FUNCTION TryConvert_USINT_TO_DWORD : BOOL
VAR_INPUT
	in : USINT;
	out : REFERENCE TO DWORD;
END_VAR

out := USINT_TO_DWORD(in);
TryConvert_USINT_TO_DWORD := TRUE;

END_FUNCTION

(* stored: Version 1.1.0.1, ProductVersion 3.1.4024.12
   POU TryConvert_USINT_TO_DWORD: Id {d2170122-908f-49f8-91d7-bdd9645c9ec2}, SpecialFunc None *)
